FUNCTION_BLOCK FB_ROB_AMR EXTENDS FB_ROB IMPLEMENTS  ITF_BA_AMR, ITF_2_AMR
VAR_INPUT
END_VAR
VAR_OUTPUT
END_VAR
VAR
		tcppos, tcpvel : stPose2D;
	jointpos, jointvel: stJoint2;
END_VAR

{warning 'Add method implementation '}
METHOD M_Dock : BOOL
END_METHOD

{error 'Add method implementation or delete method to use base implementation'}
METHOD MC_ChangeSpeedOverride : INT
VAR_INPUT
	factor	: REAL;
END_VAR
END_METHOD

{error 'Add method implementation or delete method to use base implementation'}
METHOD MC_MoveAxesAbsolute : BOOL
VAR_INPUT
	target	: stTarget3D;
END_VAR
END_METHOD

{error 'Add method implementation or delete method to use base implementation'}
METHOD MC_MoveAxesRelative : BOOL
VAR_INPUT
	axes	: ARRAY [1..6] OF FB_Axis;
	offsets	: ARRAY [1..6] OF REAL;
END_VAR
END_METHOD

{error 'Add method implementation or delete method to use base implementation'}
METHOD MC_MoveLinearAbsolute : BOOL
VAR_INPUT
	target	: stTarget3D;
END_VAR
END_METHOD

{error 'Add method implementation or delete method to use base implementation'}
METHOD MC_ReadAnalogInput : LREAL
VAR_INPUT
	input	: INT;
END_VAR
END_METHOD

{error 'Add method implementation or delete method to use base implementation'}
METHOD MC_ReadDigitalInput : BOOL
VAR_INPUT
	input	: INT;
END_VAR
END_METHOD

{error 'Add method implementation or delete method to use base implementation'}
METHOD MC_SetDigitalOutput : BOOL
VAR_INPUT
	output	: INT;
	value	: BOOL;
END_VAR
END_METHOD

{error 'Add method implementation or delete method to use base implementation'}
METHOD MC_SetOperationMode : BOOL
VAR_INPUT
	mode	: eMode;
END_VAR
END_METHOD

{warning 'Add property implementation'}
PROPERTY P_ActualAxisPos : stJoint2
GET
P_ActualAxisPos:= jointpos;
END_GET
END_PROPERTY

{warning 'Add property implementation'}
PROPERTY P_ActualJointVelocity : stJoint2
GET
P_ActualJointVelocity:= jointvel;
END_GET
END_PROPERTY

{warning 'Add property implementation'}
PROPERTY P_ActualTCPPos : stPose2D
GET
P_ActualTCPPos:=tcppos;
END_GET
END_PROPERTY

{warning 'Add property implementation'}
PROPERTY P_ActualTCPVelocity : stPose2D
GET
P_ActualTCPVelocity:=tcpvel;
END_GET
END_PROPERTY

{warning 'Add property implementation'}
PROPERTY P_IsDocked : BOOL
GET
END_GET
END_PROPERTY

{warning 'Add property implementation'}
PROPERTY P_RobotModel : STRING
GET
END_GET
END_PROPERTY

{error 'Add property implementation or delete property to use base implementation'}
PROPERTY P_TargetReached : BOOL
GET
END_GET
END_PROPERTY

END_FUNCTION_BLOCK

(* stored: Version 1.1.0.1, ProductVersion 3.1.4026.18
   POU FB_ROB_AMR: Id {cf71feff-3eb8-4d62-9de2-ec89e7c3ba43}, SpecialFunc None
   Method M_Dock: Id {6f4fe9bb-99c9-44dc-8631-d609ed742588}
   Method MC_ChangeSpeedOverride: Id {ec7d2ac7-54e7-49b1-9975-0da4040fc5c7}
   Method MC_MoveAxesAbsolute: Id {a90fe26a-f8d4-4109-9b99-ff87c07c54b3}
   Method MC_MoveAxesRelative: Id {af766e40-7eaf-4eef-8e57-0f1058f3617b}
   Method MC_MoveLinearAbsolute: Id {234e030e-1187-45c8-8047-030681912149}
   Method MC_ReadAnalogInput: Id {6b565cab-80a6-4988-bcde-de338ccce79e}
   Method MC_ReadDigitalInput: Id {a05cb14f-4d63-48c7-8ac1-2fd6f968d662}
   Method MC_SetDigitalOutput: Id {ec5804a6-fa06-4409-b993-6657f2549352}
   Method MC_SetOperationMode: Id {63c18e2b-9af6-4694-9119-714bd7c11224}
   Property P_ActualAxisPos: Id {a9bb0008-2bc7-471b-b7cd-69232649304e}
   Get Get: Id {c40e1322-8cf0-4659-99cb-1ad8b6629bcb}
   Property P_ActualJointVelocity: Id {0493ea03-284e-4697-b6d9-85f06afe56ed}
   Get Get: Id {6f83ad7c-bb1b-49e3-a3b5-2da802613af4}
   Property P_ActualTCPPos: Id {5f2eea29-65d5-4ce1-8b21-86b7c8473be6}
   Get Get: Id {fa0df135-1f19-4fd2-b0d5-1f3480c883d6}
   Property P_ActualTCPVelocity: Id {353dfdcb-eeca-4ed7-9a9e-990541ee5c2e}
   Get Get: Id {edff15a4-fbcc-4630-ae2a-c4883c3e01f6}
   Property P_IsDocked: Id {b1223d7e-f467-499a-a850-c3753fbde900}
   Get Get: Id {4fc975e3-63b2-4f01-8d05-8125246e628b}
   Property P_RobotModel: Id {c33f1393-da5c-4511-9824-46618d3ff11f}
   Get Get: Id {5e9348c1-3c06-45d0-96da-a44f08e32347}
   Property P_TargetReached: Id {1ffd5e85-127b-44be-a405-ac0615b395e0}
   Get Get: Id {57de425a-d48b-4d0b-8603-0f3a7e17fce2} *)
